PROGRAM MAIN
VAR
	stWorker_1		: ST_WORKER_VARIABLES;
	stRecipe		: ST_RECIPE_VARIABLES;
	
	// Slave positions for the cam table
	// Array [1..4] are slaves 1 - 4, each of the slave is a 2d array **REQUIRED by cam table ref**
	// Array [0..359] are master-slave position pair
	ALL_CAM			: ARRAY [1..4] OF ARRAY [0..359] OF ARRAY [0..1] OF LREAL;		
	ALL_CAM_REF		: ARRAY [1..4] OF MC_CAM_REF;		// Cam table reference
	
	nState			: INT;
	bStart			: BOOL;
	
	fbMasterCam		: FB_MasterCamControl;
	fbCamProfiles	: FB_CamProfiles;
	mcHome			: MC_Home;
	bMasterRun		: BOOL;
	bHalt			: BOOL;
	bReset			: BOOL;
	bReadDone		: BOOL;
	bCreateDone		: BOOL;
	
	bCamIn			: BOOL;
	nUpdate			: INT;
END_VAR

fbMasterCam();

CASE nState OF
	0:	// IDLE
		IF bStart THEN
			nState		:= 5;
		END_IF
	5:	// Initialize and enable the power on Master and Slaves Axes
		fbMasterCam.mInitialize(TRUE);
		IF fbMasterCam.pInitialized THEN
			fbMasterCam.mInitialize(FALSE);
			nState		:= 10;
		END_IF
	(**************** These will not be implemented in the real project ***********)
	(**************** recipe management will replace the csv file *****************)
	10:	// Read CAM profiles from CSV files and store in CAM arrays
		fbCamProfiles.mReadAndStoreSlavePositions(TRUE, ALL_CAM);
		IF fbCamProfiles.pReadDone THEN
			fbCamProfiles.mReadAndStoreSlavePositions(FALSE, ALL_CAM);
			nState		:= 15;
		END_IF
	15:	// Create Twincat digital CAM tables from CAM profile arrays
		fbCamProfiles.mCreateCamProfiles(TRUE, ALL_CAM, ALL_CAM_REF);
		IF fbCamProfiles.pCreateDone THEN
			fbCamProfiles.mCreateCamProfiles(FALSE, ALL_CAM, ALL_CAM_REF);
			GVL.rMasterVel:= 0.5;			// Start Master at minimum speed
			bMasterRun	:= TRUE;			// to couple CAM profiles
			fbMasterCam.pRunCams:= TRUE;	// Start Slaves
			nState		:= 20;
		END_IF
	(**************      ~30s to complete the csv reading     *********************)
	(******************************************************************************)
	20:	// Assign CAM tables to their respective Slave Axes
		fbMasterCam.mMultiCamIn(TRUE);
		IF fbMasterCam.pCamInDone THEN
			fbMasterCam.mMultiCamIn(TRUE);
			nState		:= 25;
		END_IF
	25:	// Speed up Master after all CAMs done coupling 
		IF NOT bMasterRun THEN
			GVL.rMasterVel	:= 180;
			bMasterRun		:= TRUE;
			nState			:= 26;
		END_IF
		
	(********************* Not used *******************)
	30:	// Stop all axes
		fbMasterCam.mHalt(bHalt);
	35: // Reset all axes
		fbMasterCam.mReset(bReset);
END_CASE
fbMasterCam.mRun(bMasterRun);

END_PROGRAM

(* stored: Version 1.1.0.1, ProductVersion 3.1.4024.15
   POU MAIN: Id {8749f6d4-9eb1-4455-8c08-9154e8b5dfe0}, SpecialFunc None *)
